// TIA Portal V16 export
// export: Created 2023-03-29T11:04:47.1539335Z, ExportSetting WithDefaults, DisplayName Totally Integrated Automation Portal, DisplayVersion V16 Update 6, DisplayName TIA Portal Version Control Interface, DisplayVersion V16 Update 2, DisplayName TIA Portal Openness, DisplayVersion V16 Update 6, DisplayName STEP 7 Professional, DisplayVersion V16 Update 6, DisplayName STEP 7 Safety, DisplayVersion V16, DisplayName WinCC Advanced, DisplayVersion V16 Update 6
DATA_BLOCK "HourWork__P2_DB"   // DB14
AUTHOR : RTecmer
FAMILY : XMHour
VERSION : 0.1
// stored: AutoNumber true, DBAccessibleFromOPCUA true, InstanceOfName godzinyPracy, InstanceOfType FB
"godzinyPracy"
   // VAR_INPUT
   //    Run_Device : Bool;
   // END_VAR
   // VAR_OUTPUT
   //    MW_hour : DWord;
   //    Sum_hour_sek : Real;
   // END_VAR
   // VAR_IN_OUT
   //    Data_sek : Int;
   //    Reset { ExternalAccessible := 'False'; ExternalVisible := 'False'; ExternalWritable := 'False'} : Bool;
   //    Data_hour : DWord;
   //    Edge_Hz { ExternalAccessible := 'False'; ExternalVisible := 'False'; ExternalWritable := 'False'} : Bool;
   // END_VAR
   // VAR
   //    sek_real { ExternalAccessible := 'False'; ExternalVisible := 'False'; ExternalWritable := 'False'} : Real;
   //    actSekReal { ExternalAccessible := 'False'; ExternalVisible := 'False'; ExternalWritable := 'False'} : Real;
   //    hour_sek { ExternalAccessible := 'False'; ExternalVisible := 'False'; ExternalWritable := 'False'} : Real;
   // END_VAR
BEGIN
END_DATA_BLOCK
